SUBAPPLICATION AUDI_E_CTUD (* Subapplication Type *)
  (* Standard: 61499-2 *)
  (* Version 1.0, 2026-06-08, franz *)
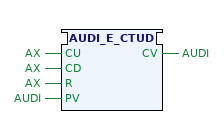
  SOCKETS
    CU : adapter::types::unidirectional::AX; (* Count Up *)
    CD : adapter::types::unidirectional::AX; (* Count Down *)
    R : adapter::types::unidirectional::AX; (* Reset *)
    PV : adapter::types::unidirectional::AUDI;
  END_SOCKETS
  PLUGS
    CV : adapter::types::unidirectional::AUDI;
  END_PLUGS
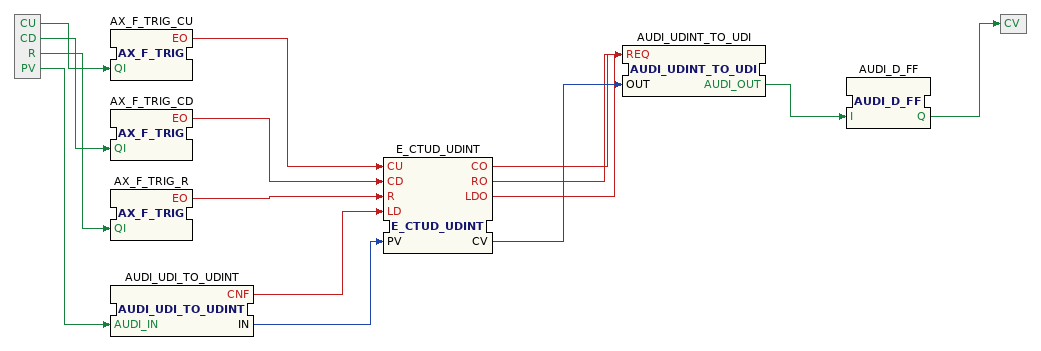
  FBS
    E_CTUD_UDINT : iec61499::events::E_CTUD_UDINT;
    AX_F_TRIG_CU : adapter::events::unidirectional::AX_F_TRIG;
    AX_F_TRIG_CD : adapter::events::unidirectional::AX_F_TRIG;
    AX_F_TRIG_R : adapter::events::unidirectional::AX_F_TRIG;
    AUDI_UDI_TO_UDINT : adapter::conversion::unidirectional::AUDI_UDI_TO_UDINT;
    AUDI_UDINT_TO_UDI : adapter::conversion::unidirectional::AUDI_UDINT_TO_UDI;
    AUDI_D_FF : adapter::events::unidirectional::AUDI_D_FF;
  END_FBS
  EVENT_CONNECTIONS
    AX_F_TRIG_CU.EO TO E_CTUD_UDINT.CU;
    AX_F_TRIG_CD.EO TO E_CTUD_UDINT.CD;
    AX_F_TRIG_R.EO TO E_CTUD_UDINT.R;
    AUDI_UDI_TO_UDINT.CNF TO E_CTUD_UDINT.LD;
    E_CTUD_UDINT.CO TO AUDI_UDINT_TO_UDI.REQ;
    E_CTUD_UDINT.RO TO AUDI_UDINT_TO_UDI.REQ;
    E_CTUD_UDINT.LDO TO AUDI_UDINT_TO_UDI.REQ;
  END_CONNECTIONS
  DATA_CONNECTIONS
    AUDI_UDI_TO_UDINT.IN TO E_CTUD_UDINT.PV;
    E_CTUD_UDINT.CV TO AUDI_UDINT_TO_UDI.OUT;
  END_CONNECTIONS
  ADAPTER_CONNECTIONS
    CU TO AX_F_TRIG_CU.QI;
    CD TO AX_F_TRIG_CD.QI;
    R TO AX_F_TRIG_R.QI;
    AUDI_D_FF.Q TO CV;
    PV TO AUDI_UDI_TO_UDINT.AUDI_IN;
    AUDI_UDINT_TO_UDI.AUDI_OUT TO AUDI_D_FF.I;
  END_CONNECTIONS
END_SUBAPPLICATION
